FUNCTION_BLOCK FB_Empleado
VAR_INPUT
	stEmpleado :ST_Empleado;
END_VAR
VAR_OUTPUT
END_VAR
VAR
	_Empleado : ST_Empleado;
END_VAR

PROPERTY Apellido : STRING
GET
Apellido := _Empleado.Apellido;
END_GET
SET
_Empleado.Apellido := Apellido;
END_SET
END_PROPERTY

PROPERTY CorreoElectronico : STRING
GET
CorreoElectronico := _Empleado.CorreoElectronico;
END_GET
SET
 _Empleado.CorreoElectronico := CorreoElectronico;
END_SET
END_PROPERTY

METHOD FB_init : BOOL
VAR_INPUT
	bInitRetains : BOOL; // if TRUE, the retain variables are initialized (warm start / cold start)
	bInCopyCode : BOOL;  // if TRUE, the instance afterwards gets moved into the copy code (online change)
	Empleado : ST_Empleado;
END_VAR
_Empleado := Empleado;
END_METHOD

PROPERTY Nombre : STRING
GET
Nombre := _Empleado.Nombre;
END_GET
SET
_Empleado.Nombre := Nombre;
END_SET
END_PROPERTY

END_FUNCTION_BLOCK

(* stored: Version 1.1.0.1, ProductVersion 3.1.4024.12
   POU FB_Empleado: Id {c9fd69cc-780b-4a7a-a81b-af4317d13695}, SpecialFunc None
   Property Apellido: Id {85706286-c597-4857-bdc8-6d087f1f29cf}
   Get Get: Id {45b57335-d209-4f38-af38-4791567ee3ee}
   Set Set: Id {4d076d00-5585-41bb-80ae-8ea9360956af}
   Property CorreoElectronico: Id {8257975b-dcfb-4072-a80e-c0f8eb6026c8}
   Get Get: Id {517e03be-b975-40a6-9d03-7c6fc7b5b0ec}
   Set Set: Id {c6ba564a-f30c-4647-82a9-c98740b45dbc}
   Method FB_init: Id {9d71571a-656c-457b-9264-3ac55785932d}
   Property Nombre: Id {4b908c39-db30-4c4c-b242-536d051266a4}
   Get Get: Id {7bf5646e-0e4b-4e19-a0ee-a53cf0b22ea3}
   Set Set: Id {7bc25f2e-1d63-4610-80a8-c90608bdc659} *)
